TYPE ST_RcvDpDevData :
STRUCT
	bAckRei		: BOOL;
	bSub00		: BOOL;
	bSub01		: BOOL;
	bSub02		: BOOL;
	bSub03		: BOOL;
	bSub04		: BOOL;
	bSub05		: BOOL;
	bSub06		: BOOL;
	bSub07		: BOOL;
	bSub08		: BOOL;
	bSub09		: BOOL;
	bSub10		: BOOL;
	bSub11		: BOOL;
	bSub12		: BOOL;
	bSub13		: BOOL;
	bSub14		: BOOL;
	bSub15		: BOOL;
	nSub00		: INT;
	nSub01		: INT;
END_STRUCT
END_TYPE

(* stored: Version 1.1.0.1, ProductVersion 3.1.4024.12
   DUT ST_RcvDpDevData: Id {11eee295-ee79-03ad-3aae-4c916fef7a70} *)
